LIN {X 0,Y 60.848,Z 232.987,A -85,B 0,C 180,E1 -29531.665,E2 -29531.665} C_VEL
LIN {X 0,Y 61.497,Z 235.802,A -85,B 0,C 180,E1 -29534.904,E2 -29534.904} C_VEL
LIN {X 0,Y 62.334,Z 242.804,A -85,B 0,C 180,E1 -29541.501,E2 -29541.501} C_VEL
LIN {X 0,Y 62.619,Z 248.773,A -85,B 0,C 180,E1 -29546.679,E2 -29546.679} C_VEL
LIN {X 0,Y 60.3,Z 257.214,A -85,B 0,C 180,E1 -29552.331,E2 -29552.331} C_VEL
LIN {X 0,Y 57.125,Z 267.094,A -85,B 0,C 180,E1 -29560.265,E2 -29560.265} C_VEL
LIN {X 0,Y 56.492,Z 268.684,A -85,B 0,C 180,E1 -29561.719,E2 -29561.719} C_VEL
LIN {X 0,Y 50.346,Z 278.077,A -85,B 0,C 180,E1 -29571.086,E2 -29571.086} C_VEL
LIN {X 0,Y 45.627,Z 285.572,A -85,B 0,C 180,E1 -29582.479,E2 -29582.479} C_VEL
LIN {X 0,Y 43.002,Z 291.577,A -85,B 0,C 180,E1 -29595.811,E2 -29595.811} C_VEL
LIN {X 0,Y 42.54,Z 296.292,A -85,B 0,C 180,E1 -29610.002,E2 -29610.002} C_VEL
LIN {X 0,Y 42.572,Z 298.612,A -85,B 0,C 180,E1 -29619.504,E2 -29619.504} C_VEL
LIN {X 0,Y 45.258,Z 301.985,A -85,B 0,C 180,E1 -29637.768,E2 -29637.768} C_VEL
LIN {X 0,Y 51.783,Z 303.971,A -85,B 0,C 180,E1 -29652.737,E2 -29652.737} C_VEL
LIN {X 0,Y 61.225,Z 304.634,A -85,B 0,C 180,E1 -29663.471,E2 -29663.471} C_VEL
LIN {X 0,Y 72.321,Z 304.02,A -85,B 0,C 180,E1 -29671,E2 -29671} C_VEL
LIN {X 0,Y 84.368,Z 302.121,A -85,B 0,C 180,E1 -29676.396,E2 -29676.396} C_VEL
LIN {X 0,Y 90.662,Z 300.687,A -85,B 0,C 180,E1 -29678.472,E2 -29678.472} C_VEL
LIN {X 0,Y 93.463,Z 299.871,A -85,B 0,C 180,E1 -29679.942,E2 -29679.942} C_VEL
LIN {X 0,Y 80.123,Z 302.093,A -85,B 0,C 180,E1 -29684.77,E2 -29684.77} C_VEL
LIN {X 0,Y 71.59,Z 302.675,A -85,B 0,C 180,E1 -29689.028,E2 -29689.028} C_VEL
LIN {X 0,Y 63.554,Z 302.516,A -85,B 0,C 180,E1 -29694.422,E2 -29694.422} C_VEL
LIN {X 0,Y 56.241,Z 301.646,A -85,B 0,C 180,E1 -29701.352,E2 -29701.352} C_VEL
LIN {X 0,Y 49.98,Z 300.035,A -85,B 0,C 180,E1 -29710.151,E2 -29710.151} C_VEL
LIN {X 0,Y 44.098,Z 296.745,A -85,B 0,C 180,E1 -29724.822,E2 -29724.822} C_VEL
LIN {X 0,Y 41.447,Z 291.94,A -85,B 0,C 180,E1 -29742.701,E2 -29742.701} C_VEL
LIN {X 0,Y 42.181,Z 287.35,A -85,B 0,C 180,E1 -29756.406,E2 -29756.406} C_VEL
LIN {X 0,Y 44.942,Z 281.357,A -85,B 0,C 180,E1 -29769.752,E2 -29769.752} C_VEL
LIN {X 0,Y 49.78,Z 273.518,A -85,B 0,C 180,E1 -29781.882,E2 -29781.882} C_VEL
LIN {X 0,Y 55.788,Z 264.473,A -85,B 0,C 180,E1 -29791.071,E2 -29791.071} C_VEL
LIN {X 0,Y 62.355,Z 253.957,A -85,B 0,C 180,E1 -29798.098,E2 -29798.098} C_VEL
LIN {X 0,Y 63.88,Z 251.281,A -85,B 0,C 180,E1 -29799.498,E2 -29799.498} C_VEL
LIN {X 0,Y 63.837,Z 246.629,A -85,B 0,C 180,E1 -29803.674,E2 -29803.674} C_VEL
LIN {X 0,Y 63.121,Z 242.277,A -85,B 0,C 180,E1 -29808.129,E2 -29808.129} C_VEL
LIN {X 0,Y 61.707,Z 237.031,A -85,B 0,C 180,E1 -29814.344,E2 -29814.344} C_VEL
LIN {X 0,Y 59.323,Z 230.479,A -85,B 0,C 180,E1 -29823.981,E2 -29823.981} C_VEL
LIN {X 0,Y 58.018,Z 227.628,A -85,B 0,C 180,E1 -29829.654,E2 -29829.654} C_VEL
LIN {X 0,Y 56.503,Z 224.312,A -85,B 0,C 180,E1 -29838.269,E2 -29838.269} C_VEL
LIN {X 0,Y 56.086,Z 223.537,A -85,B 0,C 180,E1 -29841.21,E2 -29841.21} C_VEL
LIN {X 0,Y 55.215,Z 222.574,A -85,B 0,C 180,E1 -29849.398,E2 -29849.398} C_VEL
LIN {X 0,Y 55.016,Z 222.274,A -85,B 0,C 180,E1 -29857.47,E2 -29857.47} C_VEL
LIN {X 0,Y 55.685,Z 222.423,A -85,B 0,C 180,E1 -29865.383,E2 -29865.383} C_VEL
LIN {X 0,Y 56.888,Z 223.328,A -85,B 0,C 180,E1 -29872.907,E2 -29872.907} C_VEL
LIN {X 0,Y 57.558,Z 224.288,A -85,B 0,C 180,E1 -29876.447,E2 -29876.447} C_VEL
LIN {X 0,Y 59.322,Z 228.844,A -85,B 0,C 180,E1 -29885.377,E2 -29885.377} C_VEL
LIN {X 0,Y 59.619,Z 230.367,A -85,B 0,C 180,E1 -29887.375,E2 -29887.375} C_VEL
LIN {X 0,Y 59.435,Z 233.346,A -85,B 0,C 180,E1 -29889.836,E2 -29889.836} C_VEL
LIN {X 0,Y 56.974,Z 243.607,A -85,B 0,C 180,E1 -29896.215,E2 -29896.215} C_VEL
LIN {X 0,Y 56.822,Z 245.644,A -85,B 0,C 180,E1 -29898.087,E2 -29898.087} C_VEL
LIN {X 0,Y 56.854,Z 250.375,A -85,B 0,C 180,E1 -29902.818,E2 -29902.818} C_VEL
LIN {X 0,Y 55.151,Z 255.903,A -85,B 0,C 180,E1 -29906.873,E2 -29906.873} C_VEL
LIN {X 0,Y 51.479,Z 265.578,A -85,B 0,C 180,E1 -29915.005,E2 -29915.005} C_VEL
LIN {X 0,Y 50.694,Z 267.713,A -85,B 0,C 180,E1 -29917.143,E2 -29917.143} C_VEL
LIN {X 0,Y 46.126,Z 274.329,A -85,B 0,C 180,E1 -29923.638,E2 -29923.638} C_VEL
LIN {X 0,Y 41.146,Z 281.211,A -85,B 0,C 180,E1 -29933.288,E2 -29933.288} C_VEL
LIN {X 0,Y 37.012,Z 287.975,A -85,B 0,C 180,E1 -29947.682,E2 -29947.682} C_VEL
LIN {X 0,Y 35.488,Z 293.647,A -85,B 0,C 180,E1 -29965.409,E2 -29965.409} C_VEL
LIN {X 0,Y 35.545,Z 294.854,A -85,B 0,C 180,E1 -29970.002,E2 -29970.002} C_VEL
LIN {X 0,Y 35.689,Z 297.347,A -85,B 0,C 180,E1 -29981.359,E2 -29981.359} C_VEL
LIN {X 0,Y 39.144,Z 300.949,A -85,B 0,C 180,E1 -30002.593,E2 -30002.593} C_VEL
LIN {X 0,Y 46.823,Z 303.142,A -85,B 0,C 180,E1 -30018.635,E2 -30018.635} C_VEL
LIN {X 0,Y 57.277,Z 304.09,A -85,B 0,C 180,E1 -30029.197,E2 -30029.197} C_VEL
LIN {X 0,Y 69.158,Z 303.764,A -85,B 0,C 180,E1 -30036.152,E2 -30036.152} C_VEL
LIN {X 0,Y 75.394,Z 303.106,A -85,B 0,C 180,E1 -30038.779,E2 -30038.779} C_VEL
LIN {X 0,Y 76.34,Z 302.867,A -85,B 0,C 180,E1 -30040.412,E2 -30040.412} C_VEL
LIN {X 0,Y 65.37,Z 303.178,A -85,B 0,C 180,E1 -30045.381,E2 -30045.381} C_VEL
LIN {X 0,Y 54.812,Z 302.362,A -85,B 0,C 180,E1 -30052.63,E2 -30052.63} C_VEL
LIN {X 0,Y 47.771,Z 300.97,A -85,B 0,C 180,E1 -30059.996,E2 -30059.996} C_VEL
LIN {X 0,Y 39.508,Z 297.802,A -85,B 0,C 180,E1 -30074.976,E2 -30074.976} C_VEL
LIN {X 0,Y 35.735,Z 294.633,A -85,B 0,C 180,E1 -30088.893,E2 -30088.893} C_VEL
LIN {X 0,Y 34.405,Z 289.587,A -85,B 0,C 180,E1 -30108.731,E2 -30108.731} C_VEL
LIN {X 0,Y 36.847,Z 283.25,A -85,B 0,C 180,E1 -30127.573,E2 -30127.573} C_VEL
LIN {X 0,Y 41.704,Z 275.747,A -85,B 0,C 180,E1 -30142.281,E2 -30142.281} C_VEL
LIN {X 0,Y 47.812,Z 267.337,A -85,B 0,C 180,E1 -30152.7,E2 -30152.7} C_VEL
LIN {X 0,Y 54.272,Z 258.052,A -85,B 0,C 180,E1 -30160.081,E2 -30160.081} C_VEL
LIN {X 0,Y 57.742,Z 252.637,A -85,B 0,C 180,E1 -30163.185,E2 -30163.185} C_VEL
LIN {X 0,Y 57.974,Z 250.089,A -85,B 0,C 180,E1 -30165.668,E2 -30165.668} C_VEL
LIN {X 0,Y 57.725,Z 246.827,A -85,B 0,C 180,E1 -30169.397,E2 -30169.397} C_VEL
LIN {X 0,Y 57.061,Z 243.096,A -85,B 0,C 180,E1 -30174.176,E2 -30174.176} C_VEL
LIN {X 0,Y 55.624,Z 238.005,A -85,B 0,C 180,E1 -30182.054,E2 -30182.054} C_VEL
LIN {X 0,Y 54.454,Z 234.339,A -85,B 0,C 180,E1 -30189.257,E2 -30189.257} C_VEL
LIN {X 0,Y 53.216,Z 230.821,A -85,B 0,C 180,E1 -30198.681,E2 -30198.681} C_VEL
LIN {X 0,Y 52.786,Z 229.749,A -85,B 0,C 180,E1 -30203.018,E2 -30203.018} C_VEL
LIN {X 0,Y 52.365,Z 229.255,A -85,B 0,C 180,E1 -30207.536,E2 -30207.536} C_VEL
LIN {X 0,Y 52.247,Z 228.813,A -85,B 0,C 180,E1 -30220.319,E2 -30220.319} C_VEL
LIN {X 0,Y 52.667,Z 228.875,A -85,B 0,C 180,E1 -30224.525,E2 -30224.525} C_VEL
LIN {X 0,Y 53.799,Z 229.761,A -85,B 0,C 180,E1 -30232.498,E2 -30232.498} C_VEL
LIN {X 0,Y 54.281,Z 230.967,A -85,B 0,C 180,E1 -30236.232,E2 -30236.232} C_VEL
LIN {X 0,Y 55.679,Z 235.469,A -85,B 0,C 180,E1 -30245.436,E2 -30245.436} C_VEL
LIN {X 0,Y 56.567,Z 239.28,A -85,B 0,C 180,E1 -30251.198,E2 -30251.198} C_VEL
LIN {X 0,Y 56.822,Z 245.644,A -85,B 0,C 180,E1 -30258.087,E2 -30258.087} C_VEL
LIN {X 0,Y 56.373,Z 248.169,A -85,B 0,C 180,E1 -30260.088,E2 -30260.088} C_VEL
LIN {X 0,Y 54.447,Z 251.973,A -85,B 0,C 180,E1 -30261.949,E2 -30261.949} C_VEL
LIN {X 0,Y 48.152,Z 260.536,A -85,B 0,C 180,E1 -30265.577,E2 -30265.577} C_VEL
LIN {X 0,Y 46.983,Z 262.622,A -85,B 0,C 180,E1 -30267.281,E2 -30267.281} C_VEL
LIN {X 0,Y 44.158,Z 268.465,A -85,B 0,C 180,E1 -30273.328,E2 -30273.328} C_VEL
LIN {X 0,Y 36.868,Z 277.689,A -85,B 0,C 180,E1 -30284.373,E2 -30284.373} C_VEL
LIN {X 0,Y 31.292,Z 285.01,A -85,B 0,C 180,E1 -30299.648,E2 -30299.648} C_VEL
LIN {X 0,Y 28.65,Z 290.784,A -85,B 0,C 180,E1 -30318.917,E2 -30318.917} C_VEL
LIN {X 0,Y 28.552,Z 293.353,A -85,B 0,C 180,E1 -30330.002,E2 -30330.002} C_VEL
LIN {X 0,Y 28.882,Z 295.979,A -85,B 0,C 180,E1 -30344.086,E2 -30344.086} C_VEL
LIN {X 0,Y 33.411,Z 299.838,A -85,B 0,C 180,E1 -30369.13,E2 -30369.13} C_VEL
LIN {X 0,Y 42.473,Z 302.301,A -85,B 0,C 180,E1 -30385.83,E2 -30385.83} C_VEL
LIN {X 0,Y 53.985,Z 303.477,A -85,B 0,C 180,E1 -30395.687,E2 -30395.687} C_VEL
LIN {X 0,Y 60.213,Z 303.599,A -85,B 0,C 180,E1 -30399.03,E2 -30399.03} C_VEL
LIN {X 0,Y 61.561,Z 303.565,A -85,B 0,C 180,E1 -30399.968,E2 -30399.968} C_VEL
LIN {X 0,Y 50.617,Z 302.478,A -85,B 0,C 180,E1 -30406.398,E2 -30406.398} C_VEL
LIN {X 0,Y 42.397,Z 300.798,A -85,B 0,C 180,E1 -30414.063,E2 -30414.063} C_VEL
LIN {X 0,Y 35.277,Z 298.33,A -85,B 0,C 180,E1 -30425.02,E2 -30425.02} C_VEL
LIN {X 0,Y 29.988,Z 295.087,A -85,B 0,C 180,E1 -30440.366,E2 -30440.366} C_VEL
LIN {X 0,Y 27.287,Z 289.803,A -85,B 0,C 180,E1 -30465.585,E2 -30465.585} C_VEL
LIN {X 0,Y 29.034,Z 284.486,A -85,B 0,C 180,E1 -30485.843,E2 -30485.843} C_VEL
LIN {X 0,Y 33.491,Z 277.956,A -85,B 0,C 180,E1 -30502.597,E2 -30502.597} C_VEL
LIN {X 0,Y 39.822,Z 269.995,A -85,B 0,C 180,E1 -30515.039,E2 -30515.039} C_VEL
LIN {X 0,Y 47.393,Z 260.201,A -85,B 0,C 180,E1 -30523.943,E2 -30523.943} C_VEL
LIN {X 0,Y 51.612,Z 254.227,A -85,B 0,C 180,E1 -30527.616,E2 -30527.616} C_VEL
LIN {X 0,Y 52.122,Z 253.232,A -85,B 0,C 180,E1 -30528.332,E2 -30528.332} C_VEL
LIN {X 0,Y 51.99,Z 249.055,A -85,B 0,C 180,E1 -30533.924,E2 -30533.924} C_VEL
LIN {X 0,Y 51.367,Z 244.945,A -85,B 0,C 180,E1 -30540.546,E2 -30540.546} C_VEL
LIN {X 0,Y 50.612,Z 241.01,A -85,B 0,C 180,E1 -30548.263,E2 -30548.263} C_VEL
LIN {X 0,Y 49.853,Z 238.358,A -85,B 0,C 180,E1 -30555.186,E2 -30555.186} C_VEL
LIN {X 0,Y 49.567,Z 236.772,A -85,B 0,C 180,E1 -30560.161,E2 -30560.161} C_VEL
LIN {X 0,Y 49.24,Z 235.808,A -85,B 0,C 180,E1 -30565.191,E2 -30565.191} C_VEL
LIN {X 0,Y 48.831,Z 235.223,A -85,B 0,C 180,E1 -30574.424,E2 -30574.424} C_VEL
LIN {X 0,Y 49.306,Z 235.187,A -85,B 0,C 180,E1 -30583.441,E2 -30583.441} C_VEL
LIN {X 0,Y 50.348,Z 236.062,A -85,B 0,C 180,E1 -30591.98,E2 -30591.98} C_VEL
LIN {X 0,Y 50.992,Z 239.155,A -85,B 0,C 180,E1 -30600.004,E2 -30600.004} C_VEL
LIN {X 0,Y 51.762,Z 243.391,A -85,B 0,C 180,E1 -30607.808,E2 -30607.808} C_VEL
LIN {X 0,Y 51.342,Z 250.635,A -85,B 0,C 180,E1 -30616.627,E2 -30616.627} C_VEL
LIN {X 0,Y 51.197,Z 252.48,A -85,B 0,C 180,E1 -30618.719,E2 -30618.719} C_VEL
LIN {X 0,Y 49.425,Z 257.107,A -85,B 0,C 180,E1 -30622.454,E2 -30622.454} C_VEL
LIN {X 0,Y 46.983,Z 262.622,A -85,B 0,C 180,E1 -30627.281,E2 -30627.281} C_VEL
LIN {X 0,Y 45.294,Z 265.503,A -85,B 0,C 180,E1 -30629.819,E2 -30629.819} C_VEL
LIN {X 0,Y 43.005,Z 268.233,A -85,B 0,C 180,E1 -30631.933,E2 -30631.933} C_VEL
LIN {X 0,Y 38.851,Z 272.03,A -85,B 0,C 180,E1 -30634.736,E2 -30634.736} C_VEL
LIN {X 0,Y 31.158,Z 277.813,A -85,B 0,C 180,E1 -30640.509,E2 -30640.509} C_VEL
LIN {X 0,Y 27.118,Z 281.188,A -85,B 0,C 180,E1 -30646.763,E2 -30646.763} C_VEL
LIN {X 0,Y 26.07,Z 282.298,A -85,B 0,C 180,E1 -30649.661,E2 -30649.661} C_VEL
LIN {X 0,Y 21.809,Z 289.026,A -85,B 0,C 180,E1 -30675.221,E2 -30675.221} C_VEL
LIN {X 0,Y 21.555,Z 291.765,A -85,B 0,C 180,E1 -30690.003,E2 -30690.003} C_VEL
LIN {X 0,Y 22.197,Z 294.549,A -85,B 0,C 180,E1 -30708.462,E2 -30708.462} C_VEL
LIN {X 0,Y 28.305,Z 298.644,A -85,B 0,C 180,E1 -30738.153,E2 -30738.153} C_VEL
LIN {X 0,Y 38.943,Z 301.351,A -85,B 0,C 180,E1 -30754.471,E2 -30754.471} C_VEL
LIN {X 0,Y 45.09,Z 302.242,A -85,B 0,C 180,E1 -30759.265,E2 -30759.265} C_VEL
LIN {X 0,Y 44.68,Z 302.096,A -85,B 0,C 180,E1 -30760.701,E2 -30760.701} C_VEL
LIN {X 0,Y 31.84,Z 298.666,A -85,B 0,C 180,E1 -30773.657,E2 -30773.657} C_VEL
LIN {X 0,Y 22.652,Z 293.681,A -85,B 0,C 180,E1 -30798.066,E2 -30798.066} C_VEL
LIN {X 0,Y 20.429,Z 287.657,A -85,B 0,C 180,E1 -30832.986,E2 -30832.986} C_VEL
LIN {X 0,Y 23.597,Z 282.05,A -85,B 0,C 180,E1 -30857.089,E2 -30857.089} C_VEL
LIN {X 0,Y 29.445,Z 275.263,A -85,B 0,C 180,E1 -30873.957,E2 -30873.957} C_VEL
LIN {X 0,Y 37.838,Z 265.787,A -85,B 0,C 180,E1 -30886.175,E2 -30886.175} C_VEL
LIN {X 0,Y 45.841,Z 255.71,A -85,B 0,C 180,E1 -30893.105,E2 -30893.105} C_VEL
LIN {X 0,Y 46.52,Z 253.96,A -85,B 0,C 180,E1 -30894.993,E2 -30894.993} C_VEL
LIN {X 0,Y 46.426,Z 250.409,A -85,B 0,C 180,E1 -30901.274,E2 -30901.274} C_VEL
LIN {X 0,Y 46.073,Z 246.22,A -85,B 0,C 180,E1 -30910.305,E2 -30910.305} C_VEL
LIN {X 0,Y 45.667,Z 242.516,A -85,B 0,C 180,E1 -30922.011,E2 -30922.011} C_VEL
LIN {X 0,Y 45.297,Z 241.469,A -85,B 0,C 180,E1 -30932.265,E2 -30932.265} C_VEL
LIN {X 0,Y 45.621,Z 241.339,A -85,B 0,C 180,E1 -30942.06,E2 -30942.06} C_VEL
LIN {X 0,Y 46.534,Z 242.225,A -85,B 0,C 180,E1 -30951.318,E2 -30951.318} C_VEL
LIN {X 0,Y 46.754,Z 245.507,A -85,B 0,C 180,E1 -30960.004,E2 -30960.004} C_VEL
LIN {X 0,Y 46.823,Z 248.058,A -85,B 0,C 180,E1 -30964.848,E2 -30964.848} C_VEL
LIN {X 0,Y 45.964,Z 253.648,A -85,B 0,C 180,E1 -30972.47,E2 -30972.47} C_VEL
LIN {X 0,Y 45.542,Z 255.288,A -85,B 0,C 180,E1 -30974.459,E2 -30974.459} C_VEL
LIN {X 0,Y 40.272,Z 265.33,A -85,B 0,C 180,E1 -30983.875,E2 -30983.875} C_VEL
LIN {X 0,Y 39.135,Z 267.302,A -85,B 0,C 180,E1 -30986.118,E2 -30986.118} C_VEL
LIN {X 0,Y 35,Z 272.31,A -85,B 0,C 180,E1 -30991.421,E2 -30991.421} C_VEL
LIN {X 0,Y 28.635,Z 279.355,A -85,B 0,C 180,E1 -31002.586,E2 -31002.586} C_VEL
LIN {X 0,Y 26.07,Z 282.298,A -85,B 0,C 180,E1 -31009.661,E2 -31009.661} C_VEL
LIN {X 0,Y 23.036,Z 285.356,A -85,B 0,C 180,E1 -31019.19,E2 -31019.19} C_VEL
LIN {X 0,Y 19.8,Z 287.948,A -85,B 0,C 180,E1 -31030.687,E2 -31030.687} C_VEL
LIN {X 0,Y 15.798,Z 292.168,A -85,B 0,C 180,E1 -31065.626,E2 -31065.626} C_VEL
LIN {X 0,Y 17.776,Z 294.646,A -85,B 0,C 180,E1 -31091.333,E2 -31091.333} C_VEL
LIN {X 0,Y 24.195,Z 297.399,A -85,B 0,C 180,E1 -31110.632,E2 -31110.632} C_VEL
LIN {X 0,Y 30.096,Z 299.045,A -85,B 0,C 180,E1 -31119.086,E2 -31119.086} C_VEL
LIN {X 0,Y 29.867,Z 298.934,A -85,B 0,C 180,E1 -31120.268,E2 -31120.268} C_VEL
LIN {X 0,Y 18.504,Z 294.175,A -85,B 0,C 180,E1 -31139.989,E2 -31139.989} C_VEL
LIN {X 0,Y 13.188,Z 288.191,A -85,B 0,C 180,E1 -31185.064,E2 -31185.064} C_VEL
LIN {X 0,Y 17.266,Z 281.572,A -85,B 0,C 180,E1 -31226.2,E2 -31226.2} C_VEL
LIN {X 0,Y 25.361,Z 273.674,A -85,B 0,C 180,E1 -31246.085,E2 -31246.085} C_VEL
LIN {X 0,Y 34.377,Z 264.436,A -85,B 0,C 180,E1 -31255.91,E2 -31255.91} C_VEL
LIN {X 0,Y 40.615,Z 257.172,A -85,B 0,C 180,E1 -31260.105,E2 -31260.105} C_VEL
LIN {X 0,Y 41.144,Z 256.318,A -85,B 0,C 180,E1 -31260.825,E2 -31260.825} C_VEL
LIN {X 0,Y 41.312,Z 253.039,A -85,B 0,C 180,E1 -31268.12,E2 -31268.12} C_VEL
LIN {X 0,Y 41.397,Z 251.257,A -85,B 0,C 180,E1 -31272.77,E2 -31272.77} C_VEL
LIN {X 0,Y 41.431,Z 248.907,A -85,B 0,C 180,E1 -31280.927,E2 -31280.927} C_VEL
LIN {X 0,Y 41.332,Z 247.727,A -85,B 0,C 180,E1 -31289.334,E2 -31289.334} C_VEL
LIN {X 0,Y 41.613,Z 247.307,A -85,B 0,C 180,E1 -31300.264,E2 -31300.264} C_VEL
LIN {X 0,Y 42.35,Z 248.173,A -85,B 0,C 180,E1 -31310.453,E2 -31310.453} C_VEL
LIN {X 0,Y 42.208,Z 249.772,A -85,B 0,C 180,E1 -31315.229,E2 -31315.229} C_VEL
LIN {X 0,Y 42.059,Z 251.759,A -85,B 0,C 180,E1 -31320.005,E2 -31320.005} C_VEL
LIN {X 0,Y 40.681,Z 256.587,A -85,B 0,C 180,E1 -31327.45,E2 -31327.45} C_VEL
LIN {X 0,Y 35.584,Z 264.969,A -85,B 0,C 180,E1 -31335.677,E2 -31335.677} C_VEL
LIN {X 0,Y 33.456,Z 267.953,A -85,B 0,C 180,E1 -31339.042,E2 -31339.042} C_VEL
LIN {X 0,Y 25.889,Z 275.656,A -85,B 0,C 180,E1 -31348.087,E2 -31348.087} C_VEL
LIN {X 0,Y 18.169,Z 283.168,A -85,B 0,C 180,E1 -31367.401,E2 -31367.401} C_VEL
LIN {X 0,Y 14.54,Z 289.152,A -85,B 0,C 180,E1 -31402.666,E2 -31402.666} C_VEL
LIN {X 0,Y 14.876,Z 291.563,A -85,B 0,C 180,E1 -31422.955,E2 -31422.955} C_VEL
LIN {X 0,Y 17.776,Z 294.646,A -85,B 0,C 180,E1 -31451.333,E2 -31451.333} C_VEL
LIN {X 0,Y 17.856,Z 294.844,A -85,B 0,C 180,E1 -31455.931,E2 -31455.931} C_VEL
LIN {X 0,Y 16.591,Z 294.483,A -85,B 0,C 180,E1 -31463.684,E2 -31463.684} C_VEL
LIN {X 0,Y 13.466,Z 293.138,A -85,B 0,C 180,E1 -31475.628,E2 -31475.628} C_VEL
LIN {X 0,Y 10.964,Z 291.804,A -85,B 0,C 180,E1 -31485.719,E2 -31485.719} C_VEL
LIN {X 0,Y 6.216,Z 286.971,A -85,B 0,C 180,E1 -31548.415,E2 -31548.415} C_VEL
LIN {X 0,Y 11.484,Z 281.308,A -85,B 0,C 180,E1 -31603.367,E2 -31603.367} C_VEL
LIN {X 0,Y 20.986,Z 273.546,A -85,B 0,C 180,E1 -31620.151,E2 -31620.151} C_VEL
LIN {X 0,Y 30.801,Z 264.29,A -85,B 0,C 180,E1 -31626.792,E2 -31626.792} C_VEL
LIN {X 0,Y 35.726,Z 258.95,A -85,B 0,C 180,E1 -31628.834,E2 -31628.834} C_VEL
LIN {X 0,Y 36.255,Z 257.781,A -85,B 0,C 180,E1 -31630.868,E2 -31630.868} C_VEL
LIN {X 0,Y 36.63,Z 256.062,A -85,B 0,C 180,E1 -31636.029,E2 -31636.029} C_VEL
LIN {X 0,Y 36.829,Z 255.079,A -85,B 0,C 180,E1 -31639.755,E2 -31639.755} C_VEL
LIN {X 0,Y 36.987,Z 254.019,A -85,B 0,C 180,E1 -31645.254,E2 -31645.254} C_VEL
LIN {X 0,Y 37.376,Z 253.086,A -85,B 0,C 180,E1 -31660.075,E2 -31660.075} C_VEL
LIN {X 0,Y 37.787,Z 253.915,A -85,B 0,C 180,E1 -31669.287,E2 -31669.287} C_VEL
LIN {X 0,Y 37.357,Z 255.708,A -85,B 0,C 180,E1 -31674.608,E2 -31674.608} C_VEL
LIN {X 0,Y 35.965,Z 258.797,A -85,B 0,C 180,E1 -31680.006,E2 -31680.006} C_VEL
LIN {X 0,Y 30.125,Z 266.634,A -85,B 0,C 180,E1 -31687.488,E2 -31687.488} C_VEL
LIN {X 0,Y 25.092,Z 271.61,A -85,B 0,C 180,E1 -31691.397,E2 -31691.397} C_VEL
LIN {X 0,Y 15.357,Z 279.828,A -85,B 0,C 180,E1 -31703.765,E2 -31703.765} C_VEL
LIN {X 0,Y 8.586,Z 285.769,A -85,B 0,C 180,E1 -31737.065,E2 -31737.065} C_VEL
LIN {X 0,Y 7.928,Z 289.343,A -85,B 0,C 180,E1 -31785.942,E2 -31785.942} C_VEL
LIN {X 0,Y 10.649,Z 291.766,A -85,B 0,C 180,E1 -31818.676,E2 -31818.676} C_VEL
LIN {X 0,Y 15.285,Z 293.897,A -85,B 0,C 180,E1 -31836.88,E2 -31836.88} C_VEL
LIN {X 0,Y 15.122,Z 293.805,A -85,B 0,C 180,E1 -31838.37,E2 -31838.37} C_VEL
LIN {X 0,Y 6.182,Z 287.348,A -85,B 0,C 180,E1 -31902.023,E2 -31902.023} C_VEL
LIN {X 0,Y 11.484,Z 281.308,A -85,B 0,C 180,E1 -31963.367,E2 -31963.367} C_VEL
LIN {X 0,Y 13.912,Z 279.055,A -85,B 0,C 180,E1 -31973.005,E2 -31973.005} C_VEL
LIN {X 0,Y 17.473,Z 275.11,A -85,B 0,C 180,E1 -31988.093,E2 -31988.093} C_VEL
LIN {X 0,Y 21.603,Z 270.841,A -85,B 0,C 180,E1 -31997.953,E2 -31997.953} C_VEL
LIN {X 0,Y 24.471,Z 268.087,A -85,B 0,C 180,E1 -31999.83,E2 -31999.83} C_VEL
LIN {X 0,Y 31.195,Z 261.39,A -85,B 0,C 180,E1 -32000.037,E2 -32000.037} C_VEL
LIN {X 0,Y 32.175,Z 259.89,A -85,B 0,C 180,E1 -32003.89,E2 -32003.89} C_VEL
LIN {X 0,Y 32.454,Z 258.932,A -85,B 0,C 180,E1 -32014.343,E2 -32014.343} C_VEL
LIN {X 0,Y 32.854,Z 259.488,A -85,B 0,C 180,E1 -32027.654,E2 -32027.654} C_VEL
LIN {X 0,Y 32.113,Z 260.736,A -85,B 0,C 180,E1 -32030.122,E2 -32030.122} C_VEL
LIN {X 0,Y 28.291,Z 265.248,A -85,B 0,C 180,E1 -32033.526,E2 -32033.526} C_VEL
LIN {X 0,Y 26.462,Z 267.17,A -85,B 0,C 180,E1 -32034.826,E2 -32034.826} C_VEL
LIN {X 0,Y 17.608,Z 274.792,A -85,B 0,C 180,E1 -32036.174,E2 -32036.174} C_VEL
LIN {X 0,Y 6.821,Z 282.378,A -85,B 0,C 180,E1 -32040.03,E2 -32040.03} C_VEL
LIN {X 0,Y 2.985,Z 284.694,A -85,B 0,C 180,E1 -32047.451,E2 -32047.451} C_VEL
LIN {X 0,Y 1.187,Z 285.568,A -85,B 0,C 180,E1 -32040.175,E2 -32040.175} C_VEL
LIN {X 0,Y 11.015,Z 279.05,A -85,B 0,C 180,E1 -32000.38,E2 -32000.38} C_VEL
LIN {X 0,Y 21.726,Z 270.567,A -85,B 0,C 180,E1 -31999.699,E2 -31999.699} C_VEL
LIN {X 0,Y 24.471,Z 268.087,A -85,B 0,C 180,E1 -31999.83,E2 -31999.83} C_VEL
LIN {X 0,Y 27.825,Z 269.558,A -85,B 0,C 180,E1 -31999.958,E2 -31999.958} C_VEL
LIN {X 0,Y 27.825,Z 600,A -85,B 0,C 180,E1 -31999.958,E2 -31999.958} C_VEL
LIN {X 0,Y 27.825,Z 600,A -85,B 0,C 180,E1 -31999.958,E2 -31999.958}

QRS_NEXT_CUT()

QRS_NEXT()
QRS_HOME()

END
